{attribute 'pack_mode' := '2'}
TYPE ST_MOVER_CTRL :
STRUCT
  Cmd             : E_MOVER_CTRL;  // order to execute on mover
END_STRUCT
END_TYPE

(* stored: Version 1.1.0.1
   DUT ST_MOVER_CTRL: Id {dc12ceda-02cd-42a8-af3f-4c1c9194abd0} *)
